// TIA Portal project "yxf" (V15)

(* hardware
DEVICE "S7-1200 station_1"  S7-1200 Station
   slot 0: "Rack_0"  S7-1200 Rack  Rack  V1.0
   slot 1: "PLC_1"  CPU 1214C AC/DC/Rly  6ES7 214-1BG40-0XB0  V4.2
*)

// ===== PLC "PLC_1"  CPU 1214C AC/DC/Rly =====

VAR_GLOBAL   // PLC tag table "默认变量表"
   ""on/off"" AT %I0.7 : Bool;
   ""start"" AT %I0.0 : Bool;
   ""water full"" AT %I0.1 : Bool;
   ""?????????????????"" AT %IW30 : Word;
   ""stop!!!"" AT %I0.2 : Bool;
   ""water out"" AT %I0.3 : Bool;
   ""water on"" AT %Q0.0 : Bool;
   ""run+"" AT %Q0.1 : Bool;
   ""run-"" AT %Q0.2 : Bool;
   ""water off"" AT %Q0.3 : Bool;
   ""water fuck"" AT %Q0.4 : Bool;
   ""ring"" AT %Q0.5 : Bool;
END_VAR